{attribute addProperty BoxType "EJ2914-0000-0017"}
{attribute addProperty Id "FSOEAT %I*FSOE_869360C3486"}
{attribute addProperty CRC "1958795841"}
{attribute addProperty SizeInBites "48"}
{attribute addProperty SizeInBytes "6"}
TYPE FSoE_Inputs_74C0DA41 :
STRUCT
	{attribute addProperty Name "FSOE"}
	FSOE AT %I* : FSOE_869360C3;
END_STRUCT
END_TYPE

(* stored: Version 1.2.0.0, ProductVersion 3.1.4024.9
   DUT FSoE_Inputs_74C0DA41: Id {a3ec9250-fb2c-4e1c-9735-2b7317ba50bb} *)
